(* CoDeSys 2.3.9.41 project: tok.pro *)

(* POU PLC_PRG, ST *)
PROGRAM PLC_PRG
VAR
	tok1:REAL:=4;
	tok2:REAL:=20;
	diap1,diap2 :REAL; (*диапазоны измеряемой температуры *)
	Tok : REAL ; (*ток 4-20 мА*)
	Prom : REAL ; (*промежеточная переменная*)
	lamp1: BOOL; (*лампа, выход за диапазон градусов*)
	Temp1 : REAL ; (*температура*)
END_VAR
lamp1 := (Tok > tok2) OR (Tok < tok1) ;
prom:=LIMIT(tok1, Tok, tok2);
Temp1:=((diap2*(prom-4))/16);
END_PROGRAM
